Fanuc KAREL source: kt00724.KL

-- PROVISIONAL review KL for V770-1; original PC SHA256 247f3d00509b4d693f6e0ede1ef78da2ced4d13cf1dc059f39ecdc9740d0117b
-- Incomplete behavior may be omitted. Consult companion uncertainty JSON. Do not deploy.
PROGRAM KT00724
%NOLOCKGROUP
VAR
  OUT : BOOLEAN
-- UNRESOLVED_DECL P1 type=000199
-- UNRESOLVED_DECL P2 type=000199
BEGIN
  -- UNRESOLVED_PC offsets 5-20; opcodes 22,63,23
  -- UNRESOLVED_PC offsets 25-29; opcodes 7F
END KT00724
